// TwinCAT 3 PLC project Untitled1
// ProgramVersion: 3.1.4024.0
// libraries:
//   Tc2_Standard, * (Beckhoff Automation GmbH)
//   Tc2_System, * (Beckhoff Automation GmbH)
//   Tc3_Module, * (Beckhoff Automation GmbH)
// project tree:
//   DUTs/ KOMANDA.TcDUT (not stored), POZAYZ.TcDUT (not stored), POZICIJA.TcDUT (not stored), Valj.TcDUT (not stored)
//   GVLs/ AUTO.TcGVL, GVL.TcGVL (not stored)
//   / PlcTask.TcTTO (not stored)
//   POUs/ AutoMove.TcPOU (not stored), AutoMove3.TcPOU, Counter.TcPOU (not stored), Init.TcPOU (not stored), MAIN.TcPOU (not stored), Motor.TcPOU (not stored), MotorControla.TcPOU (not stored), Multiplex.TcPOU (not stored), Automatic.TcPOU (not stored), AutoMove2.TcPOU, Motor2.TcPOU (not stored), Test.TcPOU (not stored), TrackingLogic.TcPOU (not stored)

// ---- GVLs/AUTO.TcGVL
{attribute 'qualified_only'}
VAR_GLOBAL
	Init : BOOL := FALSE;
	Varno :BOOL := FALSE;
	MotorIzbira : INT;
	VrtenjePremik : BOOL;
	VrtenjeSmer : BOOL;
	DvigPremik : BOOL;
	DvigSmer : BOOL;
	IztegPremik : BOOL;
	IztegSmer : BOOL;
	PrijemPremik : BOOL;
	PrijemSmer : BOOL;
	Current: POZICIJA;
	N: INT := 5; //v InstructionSize
	Komande0: ARRAY [0..4] OF POZICIJA := [(A := 0, Y := 0, Z := 0, P:= 0 ), 
		(A := 100, Y := 40, Z := 50, P:= 15 ),
		(A := 80, Y := 20, Z := 30, P:= 0 ),
		(A := 120, Y := 0, Z := 15, P:= 12 ),
		(A := 100, Y := 0, Z := 15, P:= 0 )];
	Status: INT := 0;
	PositionNum: INT := 2; // ne rabi
	ItemNumber : INT := 2; //ne rabi
	StageSelect : INT := 0;
	Recept : INT := 0;
	VRoki : INT := 0;
	Prijem : BOOL := FALSE;
	Positions: ARRAY [1..11] OF POZAYZ := [
			(A := 30, Y:=60, Z:= 105),
			(A := 30, Y:=60, Z:= 62),
			(A := 30, Y:=60, Z:= 20),
			(A := 60, Y:=60, Z:= 105),
			(A := 60, Y:=60, Z:= 62), // 5
			(A := 50, Y:=60, Z:= 105),
			(A := 50, Y:=60, Z:= 62),
			(A := 37, Y:=60, Z:= 105),
			(A := 40, Y:=45, Z:= 105),
			(A := 47, Y:=60, Z:= 105),
			(A := 33, Y:=0, Z:= 50)]; // 10
	Items: ARRAY [1..5] OF POZAYZ := [
			(A := 5, Y:=60, Z:= 20),
			(A := 5, Y:=60, Z:= 62),
			(A := 5, Y:=60, Z:= 105),
			(A := 50, Y:=60, Z:= 105),
			(A := 50, Y:=60, Z:= 62)];
	StageMax : INT :=10;
	Stages :  ARRAY [1 .. 3] OF ARRAY [1 .. 9] OF KOMANDA :=  [[
		(I := 1, T := 0, P := 16),
		(I := 0, T := 1, P := 0),
		(I := 2, T := 0, P := 16),
		(I := 0, T := 2, P := 0),
		(I := 3, T := 0, P := 16), // 5
		(I := 0, T := 3, P := 0),
		(I := 2, T := 0, P := 16),
		(I := 0, T := 9, P := 0),
		(I := 0, T := 11, P := 0)],
[
		(I := 5, T := 0, P := 16),
		(I := 0, T := 4, P := 0),
		(I := 4, T := 0, P := 16),
		(I := 0, T := 5, P := 0),
		(I := 4, T := 0, P := 16), // 5
		(I := 0, T := 6, P := 0),
		(I := 5, T := 0, P := 16),
		(I := 0, T := 7, P := 0),
		(I := 0, T := 11, P := 0)],
[
		(I := 1, T := 0, P := 16),
		(I := 0, T := 10, P := 0),
		(I := 2, T := 0, P := 16),
		(I := 0, T := 8, P := 0),
		(I := 3, T := 0, P := 16), // 5
		(I := 0, T := 9, P := 0),
		(I := 3, T := 0, P := 16),
		(I := 0, T := 1, P := 0),
		(I := 0, T := 11, P := 0)]];
END_VAR

// ---- POUs/AutoMove3.TcPOU
PROGRAM AutoMove3
VAR
END_VAR

END_PROGRAM

// ---- POUs/AutoMove2.TcPOU
FUNCTION_BLOCK AutoMove2
VAR_INPUT
END_VAR
VAR_OUTPUT
END_VAR
VAR
	Target : POZAYZ;
END_VAR

IF AUTO.StageSelect > 0 AND AUTO.StageSelect < AUTO.StageMax THEN
	IF AUTO.Varno = FALSE THEN
		AUTO.MotorIzbira := 3;
		AUTO.IztegSmer := TRUE;
		AUTO.IztegPremik := TRUE;
		IF AUTO.Current.Y = 0 THEN
			AUTO.Varno := TRUE;
		END_IF
	ELSIF AUTO.Stages[AUTO.Recept][Auto.StageSelect].I = 0 THEN
		Target := AUTO.Positions[AUTO.Stages[AUTO.Recept][Auto.StageSelect].T];
		IF AUTO.Current.Z <> Target.Z  THEN
			AUTO.MotorIzbira := 2;
			IF AUTO.Current.Z > Target.Z THEN
				AUTO.DvigSmer := TRUE;
			ELSE
				AUTO.DvigSmer := FALSE;
			END_IF
		AUTO.DvigPremik := TRUE;
		ELSIF AUTO.Current.A <> Target.A  THEN
			AUTO.MotorIzbira := 1;
			IF AUTO.Current.A > Target.A THEN
				AUTO.VrtenjeSmer := TRUE;
			ELSE
				AUTO.VrtenjeSmer := FALSE;
			END_IF
			AUTO.VrtenjePremik := TRUE;
		ELSIF AUTO.Current.Y <> Target.Y  THEN
			AUTO.MotorIzbira := 3;
			IF AUTO.Current.Y > Target.Y THEN
				AUTO.IztegSmer := TRUE;
			ELSE
				AUTO.IztegSmer := FALSE;
			END_IF
			AUTO.IztegPremik := TRUE;
		ELSIF AUTO.Current.P <> AUTO.Stages[AUTO.Recept][Auto.StageSelect].P  THEN
			AUTO.MotorIzbira := 4;
			IF AUTO.Current.P > AUTO.Stages[AUTO.Recept][Auto.StageSelect].P THEN
				AUTO.PrijemSmer := TRUE;
			ELSE
				AUTO.PrijemSmer := FALSE;
			END_IF
			AUTO.PrijemPremik := TRUE;
		ELSE
			AUTO.VrtenjePremik := FALSE;
			AUTO.DvigPremik := FALSE;
			AUTO.IztegPremik := FALSE;
			AUTO.PrijemPremik := FALSE;
			AUTO.StageSelect := AUTO.StageSelect + 1;
			AUTO.Varno := FALSE;
		END_IF
	ELSE
		Target := AUTO.Items[AUTO.Stages[AUTO.Recept][Auto.StageSelect].I];
			IF AUTO.Current.A <> Target.A  THEN
			AUTO.MotorIzbira := 1;
			IF AUTO.Current.A > Target.A THEN
				AUTO.VrtenjeSmer := TRUE;
			ELSE
				AUTO.VrtenjeSmer := FALSE;
			END_IF
			AUTO.VrtenjePremik := TRUE;
		ELSIF AUTO.Current.Z <> Target.Z  THEN
			AUTO.MotorIzbira := 2;
			IF AUTO.Current.Z > Target.Z THEN
				AUTO.DvigSmer := TRUE;
			ELSE
				AUTO.DvigSmer := FALSE;
			END_IF
			AUTO.DvigPremik := TRUE;
		ELSIF AUTO.Current.Y <> Target.Y  THEN
			AUTO.MotorIzbira := 3;
			IF AUTO.Current.Y > Target.Y THEN
				AUTO.IztegSmer := TRUE;
			ELSE
				AUTO.IztegSmer := FALSE;
			END_IF
			AUTO.IztegPremik := TRUE;
		ELSIF AUTO.Current.P <> AUTO.Stages[AUTO.Recept][Auto.StageSelect].P  THEN
			AUTO.MotorIzbira := 4;
			IF AUTO.Current.P > AUTO.Stages[AUTO.Recept][Auto.StageSelect].P THEN
				AUTO.PrijemSmer := TRUE;
			ELSE
				AUTO.PrijemSmer := FALSE;
			END_IF
			AUTO.PrijemPremik := TRUE;
		ELSE
			AUTO.VrtenjePremik := FALSE;
			AUTO.DvigPremik := FALSE;
			AUTO.IztegPremik := FALSE;
			AUTO.PrijemPremik := FALSE;
			AUTO.StageSelect := AUTO.StageSelect + 1;
			IF AUTO.StageSelect = AUTO.StageMax THEN
				AUTO.StageSelect := 0;
				AUTO.Init := FALSE;
				AUTO.Recept := 0;
			END_IF
			AUTO.Varno := FALSE;
		END_IF
	END_IF
	
END_IF

END_FUNCTION_BLOCK
